// TIA Portal project "Counter" (V15)

(* hardware
DEVICE "S7-1200 station_1"  S7-1200 Station
   slot 0: "Rack_0"  S7-1200 Rack  Rack  V1.0
   slot 1: "PLC_1"  CPU 1214C AC/DC/Rly  6ES7 214-1BG40-0XB0  V4.2
*)

// ===== PLC "PLC_1"  CPU 1214C AC/DC/Rly =====

VAR_GLOBAL   // PLC tag table "Default tag table"
   "Tag_1" AT %M1.1 : Bool;
   "Tag_2" AT %M1.0 : Bool;
   "Tag_3" AT %Q2.0 : Bool;
   "Tag_5" AT %M2.1 : Bool;
   "Tag_6" AT %M200.0 : Bool;
   "Tag_8" AT %MW200 : Int;
   "Tag_9" AT %MW4 : Word;
   "Tag_10" AT %MW201 : Int;
   "Tag_11" AT %MW300 : Int;
   "Tag_12" AT %M3.0 : Bool;
   "Tag_13" AT %M3.1 : Bool;
   "Tag_14" AT %M4.0 : Bool;
   "Tag_15" AT %MW400 : Int;
   "Tag_16" AT %M4.2 : Bool;
   "Tag_17" AT %M4.1 : Bool;
   "Tag_18" AT %M4.3 : Bool;
   "Tag_19" AT %MW401 : Int;
   "Tag_4" AT %M2.0 : Bool;
   "Tag_7" AT %MW402 : Int;
END_VAR

VAR_GLOBAL   // PLC tag table "Tag table_1"
   "S 1" AT %I0.0 : Bool;
   "S 2" AT %I0.1 : Bool;
   "S 3" AT %I0.2 : Bool;
   "S 4" AT %I0.3 : Bool;
   "S 5" AT %I0.4 : Bool;
   "P 1" AT %Q0.0 : Bool;
   "P 2" AT %Q0.1 : Bool;
   "P 3" AT %Q0.2 : Bool;
   "P 4" AT %Q0.3 : Bool;
   "P 5" AT %Q0.4 : Bool;
   "M 1" AT %M100.0 : Bool;
   "M 2" AT %M100.1 : Bool;
   "M 3" AT %M100.2 : Bool;
   "M 4" AT %M100.3 : Bool;
   "M 5" AT %M100.4 : Bool;
END_VAR

DATA_BLOCK "cOUNTED VALUE"   // DB2
{ S7_Optimized_Access := 'TRUE' }
VERSION : 0.1
   VAR
      "CD 1" : Int;
      "CD 2" : Int;
      "CD 3" : Int;
      "CD 4" : Int;
      "CD 5" : Int;
      "CD 6" : Int;
   END_VAR
BEGIN
END_DATA_BLOCK

// folder: System blocks/Program resources

DATA_BLOCK "CTU A"   // DB3
{ S7_Optimized_Access := 'TRUE' }
AUTHOR : Simatic
FAMILY : IEC
NAME : CNTR
VERSION : 1.0
// stored: InstanceOfName IEC_COUNTER
"IEC_COUNTER"
BEGIN
END_DATA_BLOCK

DATA_BLOCK "CTU B"   // DB4
{ S7_Optimized_Access := 'TRUE' }
AUTHOR : Simatic
FAMILY : IEC
NAME : CNTR
VERSION : 1.0
// stored: InstanceOfName IEC_COUNTER
"IEC_COUNTER"
BEGIN
END_DATA_BLOCK

DATA_BLOCK "CTU C"   // DB5
{ S7_Optimized_Access := 'TRUE' }
AUTHOR : Simatic
FAMILY : IEC
NAME : CNTR
VERSION : 1.0
// stored: InstanceOfName IEC_COUNTER
"IEC_COUNTER"
BEGIN
END_DATA_BLOCK

DATA_BLOCK "CTU D"   // DB6
{ S7_Optimized_Access := 'TRUE' }
AUTHOR : Simatic
FAMILY : IEC
NAME : CNTR
VERSION : 1.0
// stored: InstanceOfName IEC_COUNTER
"IEC_COUNTER"
BEGIN
END_DATA_BLOCK

DATA_BLOCK "CTD D"   // DB7
{ S7_Optimized_Access := 'TRUE' }
AUTHOR : Simatic
FAMILY : IEC
NAME : CNTR
VERSION : 1.0
// stored: InstanceOfName IEC_COUNTER
"IEC_COUNTER"
BEGIN
END_DATA_BLOCK

// folder: (top level)

ORGANIZATION_BLOCK "Main"   // OB1, LAD, ProgramCycle
TITLE = "Main Program Sweep (Cycle)"
{ S7_Optimized_Access := 'TRUE' }
VERSION : 0.1
   VAR_INPUT
      Initial_Call : Bool;   // Initial call of this OB
      Remanence : Bool;   // =True, if remanent data are available
   END_VAR
BEGIN

REGION Network 1: situation 1
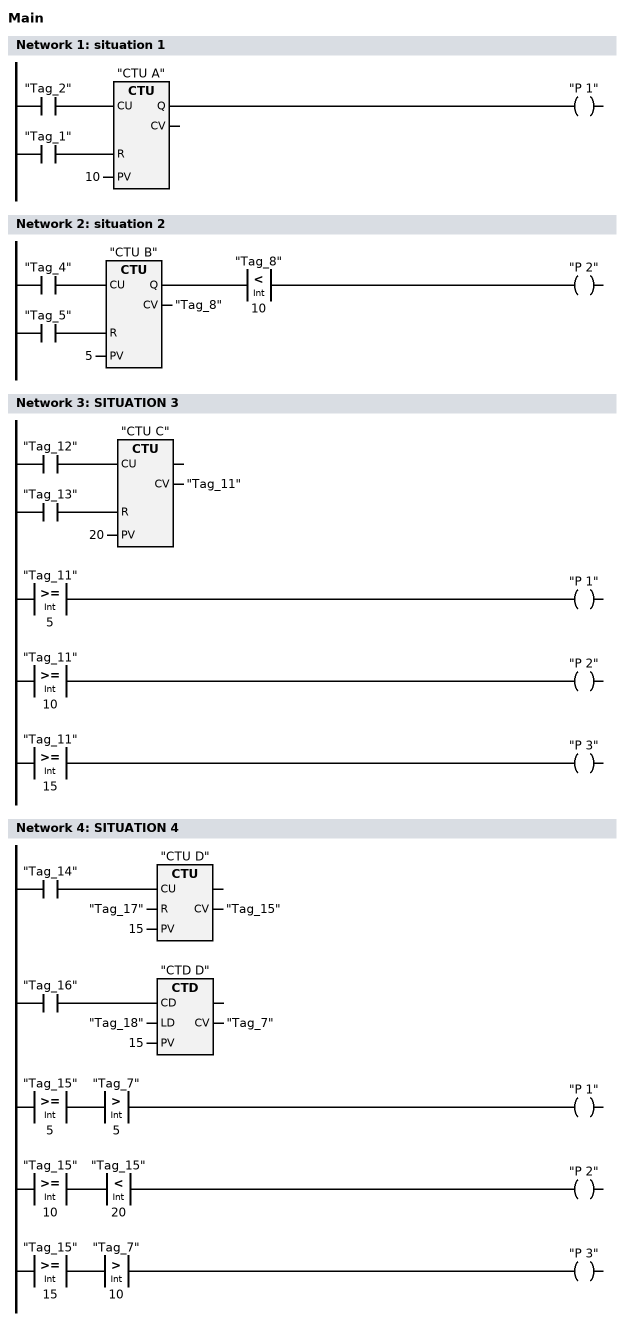
   "CTU A".CTU(CU := "Tag_2", R := "Tag_1", PV := 10);
   "P 1" := "CTU A".Q;
END_REGION

REGION Network 2: situation 2
   "CTU B".CTU(CU := "Tag_4", R := "Tag_5", PV := 5, CV => "Tag_8");
   "P 2" := "CTU B".Q AND ("Tag_8" < 10);
END_REGION

REGION Network 3: SITUATION 3
   "CTU C".CTU(CU := "Tag_12", R := "Tag_13", PV := 20, CV => "Tag_11");
   "P 1" := "Tag_11" >= 5;
   "P 2" := "Tag_11" >= 10;
   "P 3" := "Tag_11" >= 15;
END_REGION

REGION Network 4: SITUATION 4
   "CTU D".CTU(CU := "Tag_14", R := "Tag_17", PV := 15, CV => "Tag_15");
   "CTD D".CTD(CD := "Tag_16", LD := "Tag_18", PV := 15, CV => "Tag_7");
   "P 1" := ("Tag_15" >= 5) AND ("Tag_7" > 5);
   "P 2" := ("Tag_15" >= 10) AND ("Tag_15" < 20);
   "P 3" := ("Tag_15" >= 15) AND ("Tag_7" > 10);
END_REGION
END_ORGANIZATION_BLOCK